{attribute 'OPC.UA.DA' := '0'}
TYPE CanOverEthercat :
STRUCT
	AdrEthercat : UINT;
END_STRUCT
END_TYPE

(* stored: Version 1.1.0.1, ProductVersion 3.1.4024.3
   DUT CanOverEthercat: Id {ce3ffb42-f93b-4bf3-94dc-bf9391be568c} *)
